// TIA Portal V19 export
TYPE "FeedMachine_TXT"
// stored: Access Published
   STRUCT
      par_Group : String := 'Area xx Machine xx';
      Desc_P01_Man_Vel_BWD : String := 'Par01 - Velocita indietro';
      Desc_P02_Man_Vel_FWD_High : String := 'Par02 - Velocita avanti veloce';
      Desc_P03_Man_Vel_FWD_Low : String := 'Par02 - Velocita avanti lenta';
      Um_P01 : String := 'mm/min';
      Um_P02 : String := 'mm/min';
      Um_P03 : String := 'mm/min';
   END_STRUCT;
END_TYPE
